{attribute 'qualified_only'}
{attribute 'strict'}
TYPE E_DIAG_STATE :
(
	E_DIAG_DISABLED := -1,
	E_DIAG_INIT := 0,
	E_DIAG_SENDING,
	E_DIAG_WAITING
);
END_TYPE

(* stored: Version 1.1.0.1, ProductVersion 3.1.4022.12
   DUT E_DIAG_STATE: Id {f4a94788-e55b-4de1-9571-a16fdd45631e} *)
